FUNCTION_BLOCK FB_DeclineMdrConveyer IMPLEMENTS  I_MDRConveyer
VAR_INPUT
END_VAR
VAR_OUTPUT
END_VAR
VAR
	_Controller	: EP7402_REF;

	
END_VAR

METHOD Execute : BOOL
ADSLOGSTR(ADSLOG_MSGTYPE_LOG,'Moving Long-Straight','');
END_METHOD


PROPERTY MDRController : EP7402_REF
GET
MDRController := _Controller;
END_GET
SET
_Controller := MDRController;
END_SET
END_PROPERTY


METHOD Reset : BOOL
ADSLOGSTR(ADSLOG_MSGTYPE_LOG,'Reseting Long-straight','');
END_METHOD


METHOD Start : BOOL
ADSLOGSTR(ADSLOG_MSGTYPE_LOG,'Powering on Long-straight','');
END_METHOD


METHOD Stop : BOOL
ADSLOGSTR(ADSLOG_MSGTYPE_LOG,'Stopping Long-straight','');
END_METHOD

END_FUNCTION_BLOCK

(* stored: Version 1.1.0.1, ProductVersion 3.1.4024.6
   POU FB_DeclineMdrConveyer: Id {727fae8b-439f-4e2c-b09c-608ce3f3212c}, SpecialFunc None
   Method Execute: Id {1dd1545f-0666-4271-8920-ea566a687e79}
   Property MDRController: Id {c9bac534-8c4b-4ad6-a3c1-06aad1cea96c}
   Get Get: Id {5ec4a01b-8e4c-4061-a6de-b6d368336a42}
   Set Set: Id {fab36bdb-0f34-4208-9dd6-23c939e91cd3}
   Method Reset: Id {cdb775dd-a953-4044-b33c-4f59433abb84}
   Method Start: Id {1b08430a-fbfc-4cfe-932c-dc3dc8372ab4}
   Method Stop: Id {07b15d28-674e-48de-a188-11ca718c788a} *)
